(*
A list implementation for managing `I_Component`.  
*)
INTERFACE I_CompList EXTENDS I_Debug

(*
Provides the maximum capacity of the list.
*)
PROPERTY Cap : UDINT
GET
END_GET
END_PROPERTY

(*
Retrieves the `I_Component` at the specified index.  
Returns:
- `Ok` - Successfully retrieves the `I_Component`.
- `Err.Idx` - The list is empty.
- `Err.Ovf` - The specified index is out of bounds.
*)
METHOD Get : Result
VAR_INPUT
	nIndex		: UDINT;
END_VAR
VAR_OUTPUT
	iComp	: I_Component;
END_VAR
END_METHOD

(*
Returns the current number of elements in the list.
*)
PROPERTY Length : UDINT
GET
END_GET
END_PROPERTY

END_INTERFACE

(* stored: Version 1.1.0.1
   Itf I_CompList: Id {d8fd80a0-3272-49d8-a5be-503482b9faa2}
   Property Cap: Id {291c67bf-7189-4948-8947-8920d3b565a1}
   Get Get: Id {d6556997-0641-484b-bf5e-ee7b63675fab}
   Method Get: Id {6d0ac523-901f-4217-bbaf-1573baa03871}
   Property Length: Id {f505d97a-6992-4830-9f03-685b32d51775}
   Get Get: Id {f55bc4cc-b7c7-4a8d-9355-b1ef82f70d86} *)
